(* CoDeSys 2.3.9.45 project: Porte_Auto.pro *)
(* Libraries: SysLibVisu.lib 2.12.10 14:48:32, Standard.lib 2.12.10 14:48:34, SYSLIBCALLBACK.LIB 2.12.10 14:48:32 *)

(* PLC configuration (modules and I/O channels)
AT %IX0.0 [BOOLOnX_I] Ch_1 Digital input
AT %IX0.1 [BOOLOnX_I] Ch_2 Digital input
AT %IX0.2 [BOOLOnX_I] Ch_3 Digital input
AT %IX0.3 [BOOLOnX_I] Ch_4 Digital input
AT %IX0.4 [BOOLOnX_I] Ch_5 Digital input
AT %IX0.5 [BOOLOnX_I] Ch_6 Digital input
AT %IX0.6 [BOOLOnX_I] Ch_7 Digital input
AT %IX0.7 [BOOLOnX_I] Ch_8 Digital input
K1 AT %QX0.0 [BOOLOnX_Q] Ch_1 Digital output
K2 AT %QX0.1 [BOOLOnX_Q] Ch_2 Digital output
K3 AT %QX0.2 [BOOLOnX_Q] Ch_3 Digital output
K4 AT %QX0.3 [BOOLOnX_Q] Ch_4 Digital output
DEF AT %QX0.4 [BOOLOnX_Q] Ch_5 Digital output
MTN AT %QX0.5 [BOOLOnX_Q] Ch_6 Digital output
AT %QX0.6 [BOOLOnX_Q] Ch_7 Digital output
AT %QX0.7 [BOOLOnX_Q] Ch_8 Digital output
Fieldbus variables [FB_VARS] node 1, in %IB0 out %QB0
Flag variables [FLAG_VARS] node 2, in %IB0 out %QB0
Modbus-Master [MB_MASTER] node 3, in %IB0 out %QB0
*)

(* Task configuration *)
TASK cycle_2ms (PRIORITY := 0, INTERVAL := T#2ms);
	porte_atelier();
	PLC_PRG
END_TASK

(* Global variable list: Variables_Globales *)
VAR_GLOBAL
	vitesse:INT; 	(*de 0 à 10*)
	descente:INT; (*de 0 à -450*)
	FCH,FCB,MON,DES, SER,PRES :BOOL;
END_VAR

(* POU porte_atelier, CFC *)
PROGRAM porte_atelier
VAR
END_VAR
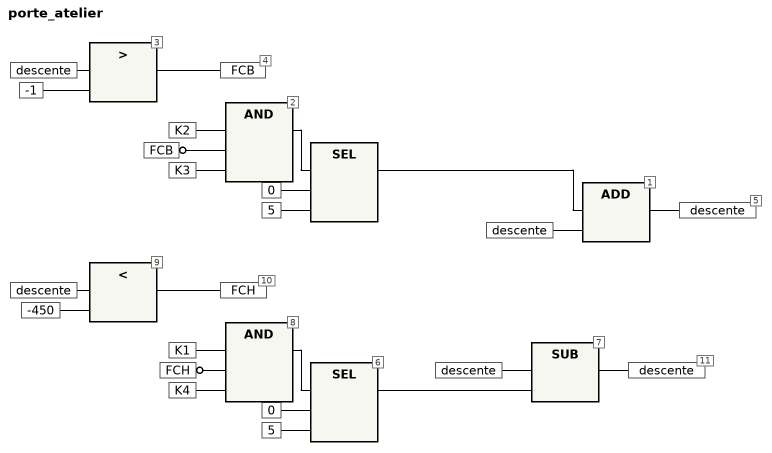
_CFC_ (* Continuous Function Chart, elements in execution order *)
#0 SEL(#2, 0, 5)
#1 ADD(#0, descente)
#2 AND(K2, NOT FCB, K3)
#3 >(descente, -1)
#4 FCB <= #3
#5 descente <= #1
#6 SEL(#8, 0, 5)
#7 SUB(descente, #6)
#8 AND(K1, NOT FCH, K4)
#9 <(descente, -450)
#10 FCH <= #9
#11 descente <= #7
_END_CFC_
END_PROGRAM

(* POU PLC_PRG, LD *)
PROGRAM PLC_PRG

VAR
	OUV: BOOL;
	t1: TON;
	cpt1: CTU;
	B_RESET: BOOL;
END_VAR
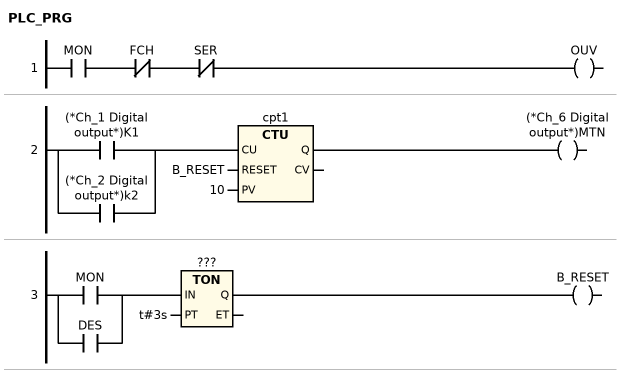
_LD_ (* Ladder Diagram *)
NETWORK 1
	[MON] - [/FCH] - [/SER] --- (OUV)
NETWORK 2
	{ [(*Ch_1 Digital output*)K1] | [(*Ch_2 Digital output*)k2] } - cpt1:CTU(CU: *, RESET: B_RESET, PV: 10) --- ((*Ch_6 Digital output*)MTN)
NETWORK 3
	{ [MON] | [DES] } - ???:TON(IN: *, PT: t#3s) --- (B_RESET)
_END_LD_
(* the same logic as Structured Text *)
(* Network 1 *)
OUV := MON AND NOT FCH AND NOT SER;
(* Network 2 *)
cpt1(CU := ((*Ch_1 Digital output*)K1) OR ((*Ch_2 Digital output*)k2), RESET := B_RESET, PV := 10);
(*Ch_6 Digital output*)MTN := cpt1.Q;
(* Network 3: see the listing above *)
END_PROGRAM

(* POU PLC_PRG_latest, FBD *)
PROGRAM PLC_PRG_latest

VAR
	OUV: BOOL;
	FER: BOOL;
	t1: TON;
	t2: TON;
	cpt1: CTU;
END_VAR
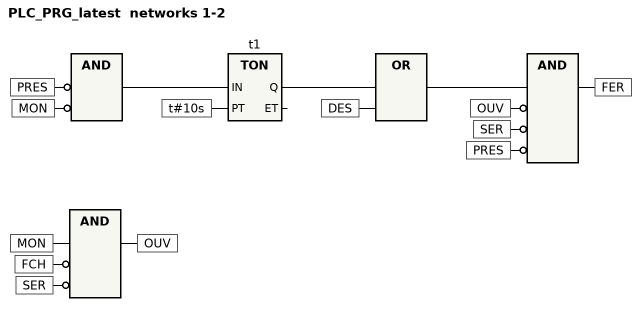
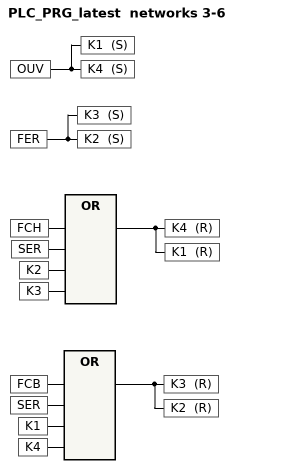
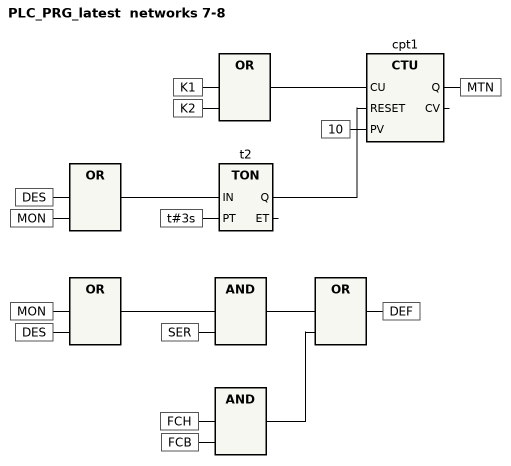
_FBD_ (* Function Block Diagram *)
NETWORK 1
	AND(OR(t1:TON(IN: AND(NOT PRES, NOT MON), PT: t#10s), DES), NOT OUV, NOT SER, NOT PRES) => FER
NETWORK 2
	AND(MON, NOT FCH, NOT SER) => OUV
NETWORK 3
	<OUV => S K1> => S K4
NETWORK 4
	<FER => S K3> => S K2
NETWORK 5
	<OR(FCH, SER, K2, K3) => R K4> => R K1
NETWORK 6
	<OR(FCB, SER, K1, K4) => R K3> => R K2
NETWORK 7
	cpt1:CTU(CU: OR(K1, K2), RESET: t2:TON(IN: OR(DES, MON), PT: t#3s), PV: 10) => MTN
NETWORK 8
	OR(AND(OR(MON, DES), SER), AND(FCH, FCB)) => DEF
_END_FBD_
(* the same logic as Structured Text *)
(* Network 1 *)
t1(IN := NOT PRES AND NOT MON, PT := t#10s);
FER := (t1.Q OR DES) AND NOT OUV AND NOT SER AND NOT PRES;
(* Network 2 *)
OUV := MON AND NOT FCH AND NOT SER;
(* Network 3 *)
IF OUV THEN K1 := TRUE; END_IF;
IF OUV THEN K4 := TRUE; END_IF;
(* Network 4 *)
IF FER THEN K3 := TRUE; END_IF;
IF FER THEN K2 := TRUE; END_IF;
(* Network 5 *)
IF FCH OR SER OR K2 OR K3 THEN K4 := FALSE; END_IF;
IF FCH OR SER OR K2 OR K3 THEN K1 := FALSE; END_IF;
(* Network 6 *)
IF FCB OR SER OR K1 OR K4 THEN K3 := FALSE; END_IF;
IF FCB OR SER OR K1 OR K4 THEN K2 := FALSE; END_IF;
(* Network 7 *)
t2(IN := DES OR MON, PT := t#3s);
cpt1(CU := K1 OR K2, RESET := t2.Q, PV := 10);
MTN := cpt1.Q;
(* Network 8 *)
DEF := ((MON OR DES) AND SER) OR (FCH AND FCB);
END_PROGRAM

(* Visualisation Entrees
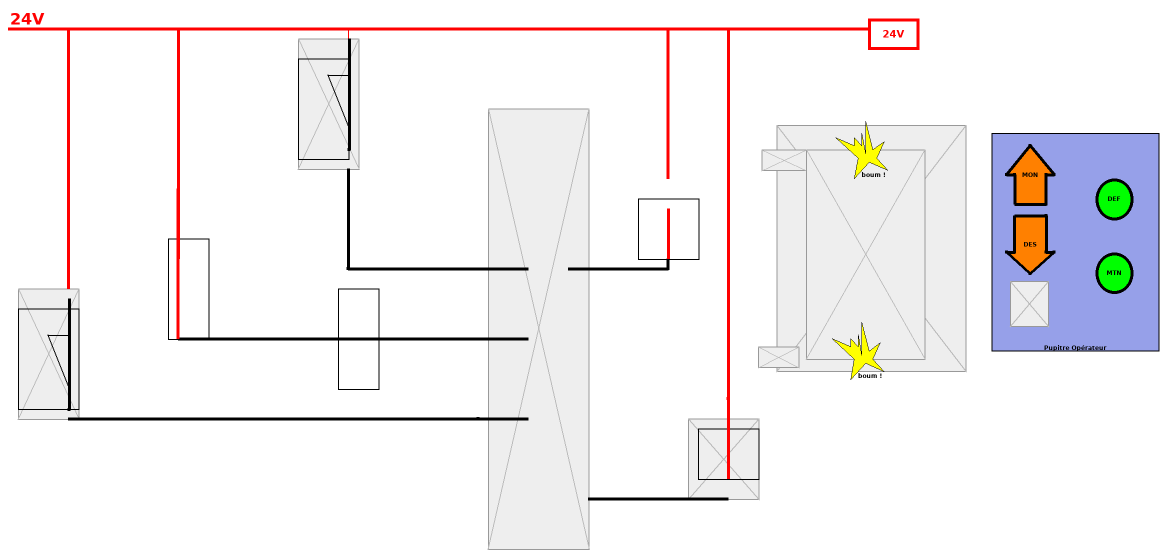
bitmap at (500,110)-(601,551): c:\users\nicolas\documents\iut 2021-2022\but\r1.07_automatisme_s1\projets_codesys\po_virtuelles\750-430.jpg
bitmap at (30,290)-(91,421): c:\users\nicolas\documents\iut 2021-2022\but\r1.07_automatisme_s1\projets_codesys\po_virtuelles\contact_fc_no.jpg
bitmap at (310,40)-(371,171): c:\users\nicolas\documents\iut 2021-2022\but\r1.07_automatisme_s1\projets_codesys\po_virtuelles\contact_fc_no.jpg
polyline at (360,170)-(540,270): alarm colour if FCB
polyline at (80,420)-(540,420): alarm colour if FCB
bitmap at (700,420)-(771,501): c:\users\nicolas\documents\iut 2021-2022\but\r1.07_automatisme_s1\projets_codesys\po_virtuelles\bp.jpg
polyline at (580,260)-(680,270): alarm colour if MON
polyline at (600,500)-(740,500): alarm colour if DES
polyline at (20,30)-(880,30): text "24V"
rectangle at (880,20)-(931,51): text "24V"
rectangle at (310,60)-(361,161): invisible if NOT(FCH)
rectangle at (30,310)-(91,411): invisible if NOT(FCB)
rectangle at (350,290)-(391,391): invisible if NOT(SER)
polyline at (190,340)-(540,340): alarm colour if SER
rectangle at (710,430)-(771,481): invisible if NOT(DES)
polyline at (740,430)-(740,480): invisible if NOT(DES)
rectangle at (650,200)-(711,261): invisible if NOT(MON)
polyline at (680,210)-(680,260): invisible if NOT(MON)
embedded screen at (770,110)-(1171,381): PO_PR
rectangle at (180,240)-(221,341): invisible if NOT(SER)
polyline at (190,240)-(190,340): invisible if NOT(SER)
9 more shapes without text or variables
2 elements of other kinds (tables, trends, ...) not read
*)

(* Visualisation PO_PR
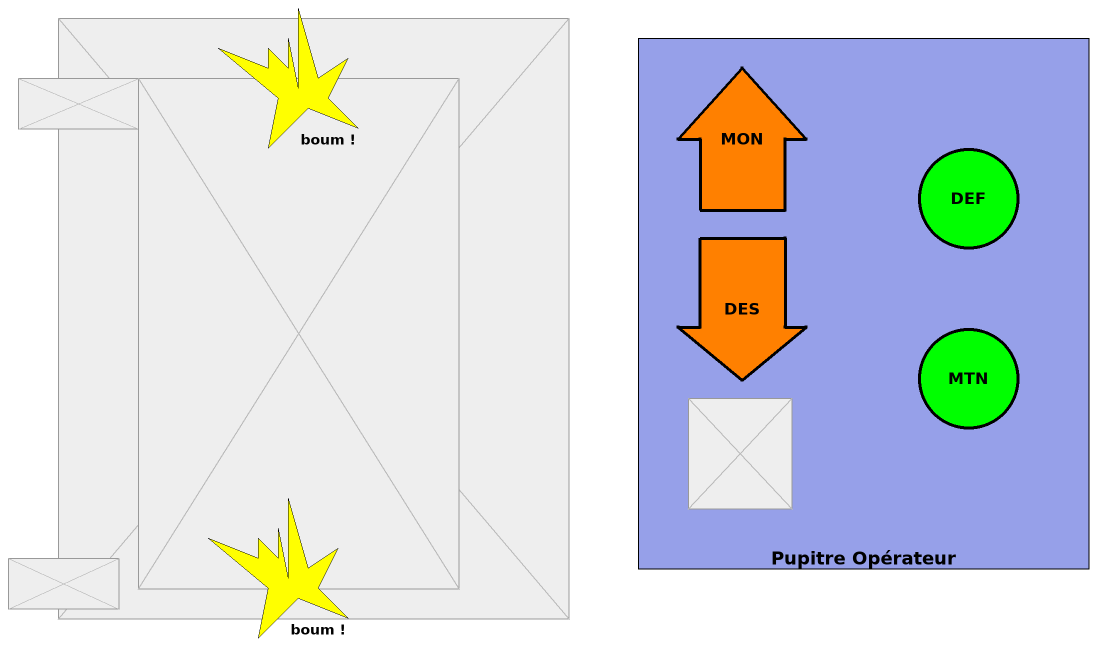
bitmap at (40,40)-(551,641): cadre_porte.jpg
bitmap at (-10,580)-(101,631): fdc.jpg
bitmap at (0,100)-(121,151): fdc.jpg
bitmap at (120,100)-(441,611): porte.jpg
rounded rectangle at (620,60)-(1071,591): text "Pupitre Opérateur"
polygon at (660,90)-(788,232): text "MON"; taps MON
polygon at (660,260)-(788,402): text "DES"; taps DES
bitmap at (670,420)-(774,531): serrure.jpg
ellipse at (900,170)-(1001,271): text "DEF"; alarm colour if DEF
ellipse at (900,350)-(1001,451): text "MTN"; alarm colour if MTN
polygon at (200,30)-(340,170): text "boum !"; invisible if NOT(FCH AND K1 AND K4)
polygon at (190,520)-(330,660): text "boum !"; invisible if NOT(FCB AND K2 AND K3)
1 more shapes without text or variables
*)

(* Visualisation schema_puiss
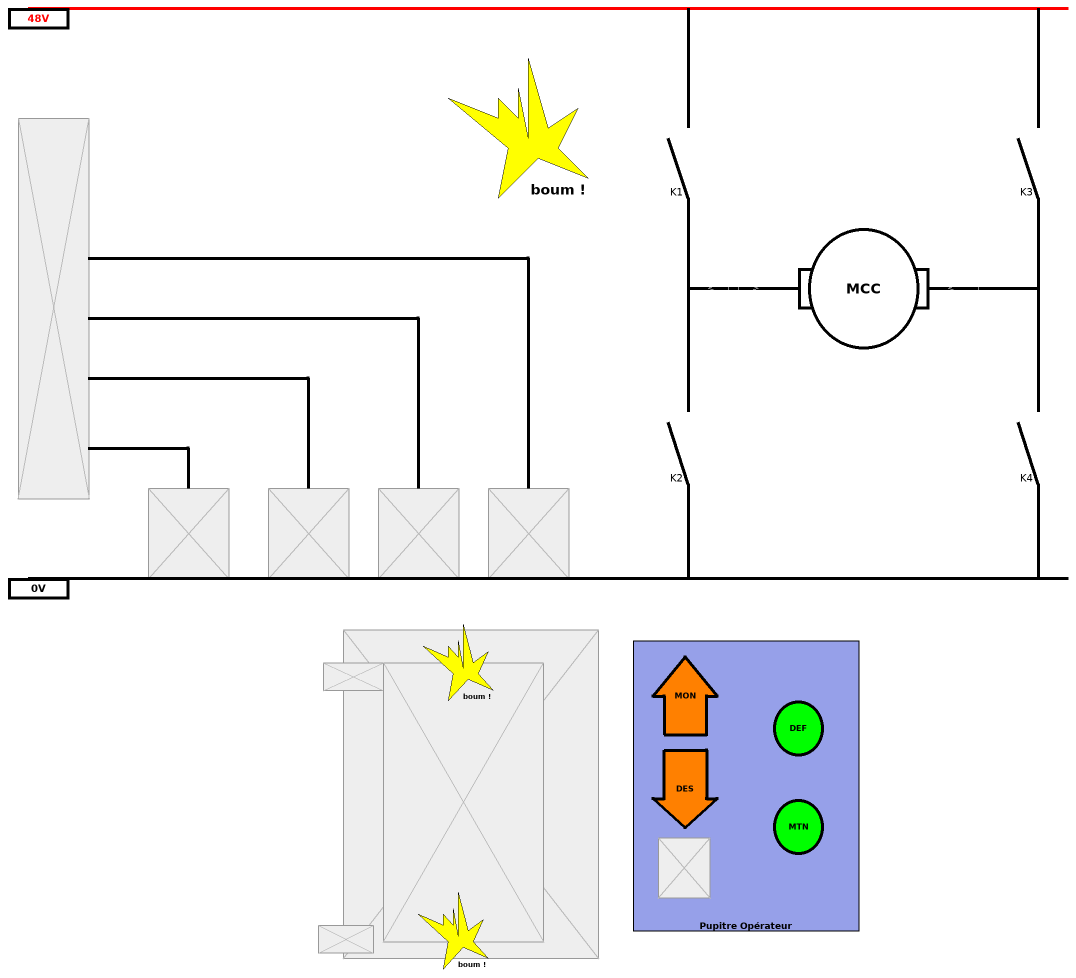
bitmap at (510,500)-(591,591): c:\users\nicolas\documents\iut 2021-2022\but\r1.07_automatisme_s1\projets_codesys\po_virtuelles\bobine_relais.jpg
bitmap at (400,500)-(481,591): c:\users\nicolas\documents\iut 2021-2022\but\r1.07_automatisme_s1\projets_codesys\po_virtuelles\bobine_relais.jpg
bitmap at (290,500)-(371,591): c:\users\nicolas\documents\iut 2021-2022\but\r1.07_automatisme_s1\projets_codesys\po_virtuelles\bobine_relais.jpg
bitmap at (170,500)-(251,591): c:\users\nicolas\documents\iut 2021-2022\but\r1.07_automatisme_s1\projets_codesys\po_virtuelles\bobine_relais.jpg
bitmap at (40,130)-(111,511): c:\users\nicolas\documents\iut 2021-2022\but\r1.07_automatisme_s1\projets_codesys\po_virtuelles\750-530.jpg
rectangle at (30,20)-(91,41): text "48V"
rectangle at (30,590)-(91,611): text "0V"
polyline at (110,460)-(210,500): alarm colour if K1
polyline at (110,390)-(330,500): alarm colour if K2
polyline at (110,330)-(440,500): alarm colour if K3
polyline at (110,270)-(550,500): alarm colour if K4
polyline at (710,300)-(820,300): alarm colour if K1 AND K4 OR K2 AND K3
polyline at (710,300)-(710,424): alarm colour if K2
polyline at (710,424)-(710,496): alarm colour if K2
polyline at (690,434)-(710,496): text "K2"; alarm colour if K2
polyline at (710,496)-(710,589): alarm colour if K2
polyline at (1060,20)-(1060,140): alarm colour if K3
polyline at (1060,140)-(1060,210): alarm colour if K3
polyline at (1040,150)-(1060,210): text "K3"; alarm colour if K3
polyline at (1060,210)-(1060,300): alarm colour if K3
polyline at (1060,300)-(1060,424): alarm colour if K4
polyline at (1060,424)-(1060,496): alarm colour if K4
polyline at (1040,434)-(1060,496): text "K4"; alarm colour if K4
polyline at (1060,496)-(1060,589): alarm colour if K4
ellipse at (830,240)-(941,361): text "MCC"
polyline at (710,20)-(710,140): alarm colour if K1
polyline at (710,140)-(710,210): alarm colour if K1
polyline at (690,150)-(710,210): text "K1"; alarm colour if K1
polyline at (710,210)-(710,300): alarm colour if K1
polygon at (750,290)-(780,310): alarm colour if K1 AND K4 AND NOT(K2) AND NOT(K3)
polygon at (980,290)-(1010,310): alarm colour if K1 AND K4 AND NOT(K2) AND NOT(K3)
polyline at (950,300)-(1060,300): alarm colour if K1 AND K4 OR K2 AND K3
polygon at (730,290)-(760,310): alarm colour if K2 AND K3 AND NOT(K1) AND NOT(K4)
polygon at (970,290)-(1000,310): alarm colour if K2 AND K3 AND NOT(K1) AND NOT(K4)
embedded screen at (340,620)-(881,981): PO_PR
polygon at (470,70)-(610,210): text "boum !"; invisible if NOT(K1 AND K2 OR K3 AND K4)
3 more shapes without text or variables
*)
